Staubli VAL3: onF7Event.pgx

program onF7Event(bool& x_bSave[])
  local string l_sMessage
  local bool l_bFound
  local string l_sTrajName
  local bool l_bYes
  local string l_sString
  local string l_sButton[2]
begin
  // look if the bButton is enable
  if bButton[6]
    // delete the selected tool

  endIf
end
